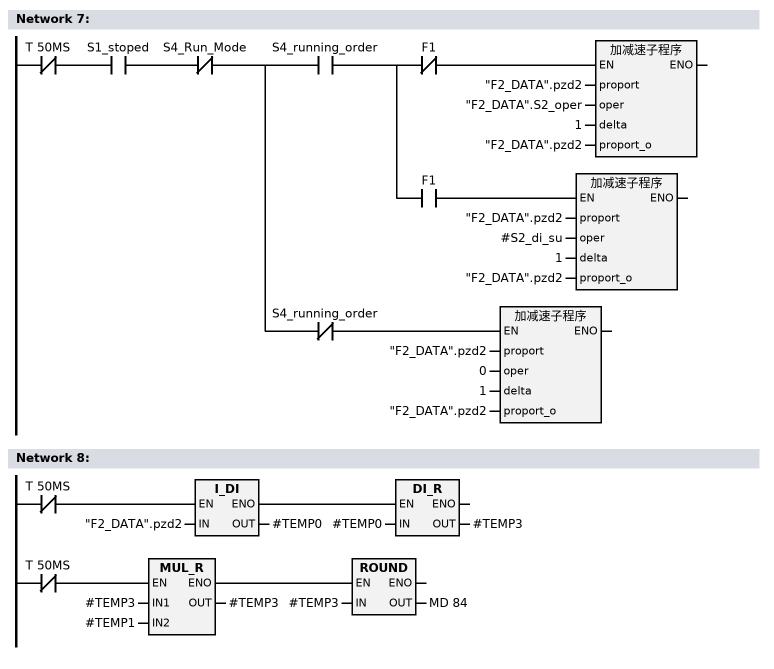
NETWORK
TITLE =
      AN    "T 50MS";
      A     "S1_stoped";
      AN    "S4_Run_Mode";
      =     L 20.0;
      A     L 20.0;
      A     "S4_running_order";
      =     L 20.1;
      A     L 20.1;
      AN    "F1";
      JNB   _00e;
      CALL  "加减速子程序" (
           proport                  := "F2_DATA".pzd2,
           oper                     := "F2_DATA".S2_oper,
           delta                    := 1,
           proport_o                := "F2_DATA".pzd2);
_00e: NOP   0;
      A     L 20.1;
      A     "F1";
      JNB   _00f;
      CALL  "加减速子程序" (
           proport                  := "F2_DATA".pzd2,
           oper                     := #S2_di_su,
           delta                    := 1,
           proport_o                := "F2_DATA".pzd2);
_00f: NOP   0;
      A     L 20.0;
      AN    "S4_running_order";
      JNB   _010;
      CALL  "加减速子程序" (
           proport                  := "F2_DATA".pzd2,
           oper                     := 0,
           delta                    := 1,
           proport_o                := "F2_DATA".pzd2);
_010: NOP   0;
NETWORK
TITLE =
      AN    "T 50MS";
      =     L 20.0;
      A(;
      A     L 20.0;
      JNB   _011;
      L     "F2_DATA".pzd2;
      ITD;
      T     #TEMP0;
      SET;
      SAVE;
      CLR;
_011: A     BR;
      );
      JNB   _012;
      L     #TEMP0;
      DTR;
      T     #TEMP3;
_012: NOP   0;
      A(;
      A     L 20.0;
      JNB   _013;
      L     #TEMP3;
      L     #TEMP1;
      *R;
      T     #TEMP3;
      AN    OV;
      SAVE;
      CLR;
_013: A     BR;
      );
      JNB   _014;
      L     #TEMP3;
      RND;
      T     MD 84;
_014: NOP   0;
END_FUNCTION

FUNCTION FC 114 : VOID
VERSION : 0.1
BEGIN
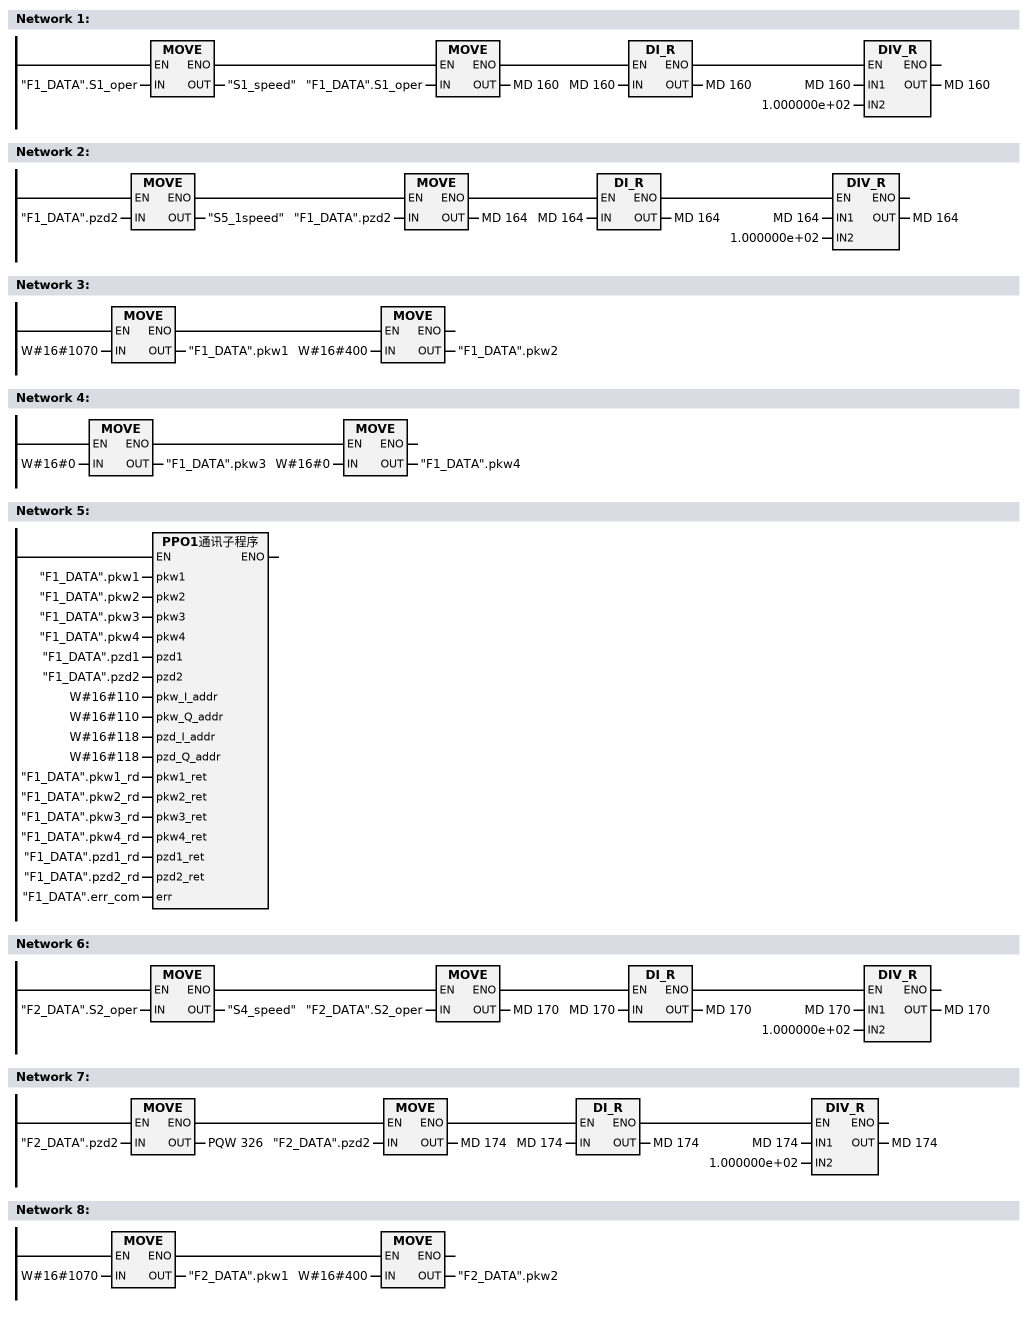
NETWORK
TITLE =
      A(;
      A(;
      A(;
      L     "F1_DATA".S1_oper;
      T     "S1_speed";
      SET;
      SAVE;
      CLR;
      A     BR;
      );
      JNB   _001;
      L     "F1_DATA".S1_oper;
      T     MD 160;
      SET;
      SAVE;
      CLR;
_001: A     BR;
      );
      JNB   _002;
      L     MD 160;
      DTR;
      T     MD 160;
      SET;
      SAVE;
      CLR;
_002: A     BR;
      );
      JNB   _003;
      L     MD 160;
      L     1.000000e+02;
      /R;
      T     MD 160;
_003: NOP   0;
NETWORK
TITLE =
      A(;
      A(;
      A(;
      L     "F1_DATA".pzd2;
      T     "S5_1speed";
      SET;
      SAVE;
      CLR;
      A     BR;
      );
      JNB   _004;
      L     "F1_DATA".pzd2;
      T     MD 164;
      SET;
      SAVE;
      CLR;
_004: A     BR;
      );
      JNB   _005;
      L     MD 164;
      DTR;
      T     MD 164;
      SET;
      SAVE;
      CLR;
_005: A     BR;
      );
      JNB   _006;
      L     MD 164;
      L     1.000000e+02;
      /R;
      T     MD 164;
_006: NOP   0;
NETWORK
TITLE =
      A(;
      L     W#16#1070;
      T     "F1_DATA".pkw1;
      SET;
      SAVE;
      CLR;
      A     BR;
      );
      JNB   _007;
      L     W#16#400;
      T     "F1_DATA".pkw2;
_007: NOP   0;
NETWORK
TITLE =
      A(;
      L     W#16#0;
      T     "F1_DATA".pkw3;
      SET;
      SAVE;
      CLR;
      A     BR;
      );
      JNB   _008;
      L     W#16#0;
      T     "F1_DATA".pkw4;
_008: NOP   0;
NETWORK
TITLE =
      CALL  "PPO1通讯子程序" (
           pkw1                     := "F1_DATA".pkw1,
           pkw2                     := "F1_DATA".pkw2,
           pkw3                     := "F1_DATA".pkw3,
           pkw4                     := "F1_DATA".pkw4,
           pzd1                     := "F1_DATA".pzd1,
           pzd2                     := "F1_DATA".pzd2,
           pkw_I_addr               := W#16#110,
           pkw_Q_addr               := W#16#110,
           pzd_I_addr               := W#16#118,
           pzd_Q_addr               := W#16#118,
           pkw1_ret                 := "F1_DATA".pkw1_rd,
           pkw2_ret                 := "F1_DATA".pkw2_rd,
           pkw3_ret                 := "F1_DATA".pkw3_rd,
           pkw4_ret                 := "F1_DATA".pkw4_rd,
           pzd1_ret                 := "F1_DATA".pzd1_rd,
           pzd2_ret                 := "F1_DATA".pzd2_rd,
           err                      := "F1_DATA".err_com);
      NOP   0;
NETWORK
TITLE =
      A(;
      A(;
      A(;
      L     "F2_DATA".S2_oper;
      T     "S4_speed";
      SET;
      SAVE;
      CLR;
      A     BR;
      );
      JNB   _009;
      L     "F2_DATA".S2_oper;
      T     MD 170;
      SET;
      SAVE;
      CLR;
_009: A     BR;
      );
      JNB   _00a;
      L     MD 170;
      DTR;
      T     MD 170;
      SET;
      SAVE;
      CLR;
_00a: A     BR;
      );
      JNB   _00b;
      L     MD 170;
      L     1.000000e+02;
      /R;
      T     MD 170;
_00b: NOP   0;
NETWORK
TITLE =
      A(;
      A(;
      A(;
      L     "F2_DATA".pzd2;
      T     PQW 326;
      SET;
      SAVE;
      CLR;
      A     BR;
      );
      JNB   _00c;
      L     "F2_DATA".pzd2;
      T     MD 174;
      SET;
      SAVE;
      CLR;
_00c: A     BR;
      );
      JNB   _00d;
      L     MD 174;
      DTR;
      T     MD 174;
      SET;
      SAVE;
      CLR;
_00d: A     BR;
      );
      JNB   _010;
      L     MD 174;
      L     1.000000e+02;
      /R;
      T     MD 174;
_010: NOP   0;
NETWORK
TITLE =
      A(;
      L     W#16#1070;
      T     "F2_DATA".pkw1;
      SET;
      SAVE;
      CLR;
      A     BR;
      );
      JNB   _011;
      L     W#16#400;
      T     "F2_DATA".pkw2;
_011: NOP   0;
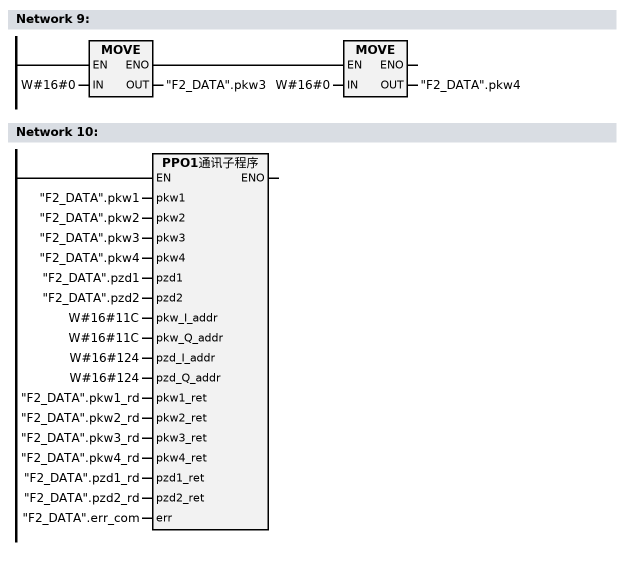
NETWORK
TITLE =
      A(;
      L     W#16#0;
      T     "F2_DATA".pkw3;
      SET;
      SAVE;
      CLR;
      A     BR;
      );
      JNB   _012;
      L     W#16#0;
      T     "F2_DATA".pkw4;
_012: NOP   0;
NETWORK
TITLE =
      CALL  "PPO1通讯子程序" (
           pkw1                     := "F2_DATA".pkw1,
           pkw2                     := "F2_DATA".pkw2,
           pkw3                     := "F2_DATA".pkw3,
           pkw4                     := "F2_DATA".pkw4,
           pzd1                     := "F2_DATA".pzd1,
           pzd2                     := "F2_DATA".pzd2,
           pkw_I_addr               := W#16#11C,
           pkw_Q_addr               := W#16#11C,
           pzd_I_addr               := W#16#124,
           pzd_Q_addr               := W#16#124,
           pkw1_ret                 := "F2_DATA".pkw1_rd,
           pkw2_ret                 := "F2_DATA".pkw2_rd,
           pkw3_ret                 := "F2_DATA".pkw3_rd,
           pkw4_ret                 := "F2_DATA".pkw4_rd,
           pzd1_ret                 := "F2_DATA".pzd1_rd,
           pzd2_ret                 := "F2_DATA".pzd2_rd,
           err                      := "F2_DATA".err_com);
      NOP   0;
END_FUNCTION

DATA_BLOCK "F1_DATA"	// DB 1
VERSION : 0.1
  STRUCT
   pkw1 : WORD  := W#16#1070;
   pkw2 : WORD  := W#16#400;
   pkw3 : WORD ;
   pkw4 : WORD ;
   pzd1 : WORD  := W#16#82;
   pzd2 : INT  := 2000;
   pkw1_rd : WORD ;
   pkw2_rd : WORD ;
   pkw3_rd : WORD ;
   pkw4_rd : WORD ;
   pzd1_rd : WORD ;
   pzd2_rd : WORD ;
   err_com : BOOL ;
   S1_oper : INT ;
  END_STRUCT ;	
BEGIN
   pkw1 := W#16#1070;
   pkw2 := W#16#400;
   pzd1 := W#16#82;
   pzd2 := 2000;
END_DATA_BLOCK

DATA_BLOCK "F2_DATA"	// DB 2
VERSION : 0.1
  STRUCT
   pkw1 : WORD ;
   pkw2 : WORD ;
   pkw3 : WORD ;
   pkw4 : WORD ;
   pzd1 : WORD ;
   pzd2 : INT ;
   pkw1_rd : WORD ;
   pkw2_rd : WORD ;
   pkw3_rd : WORD ;
   pkw4_rd : WORD ;
   pzd1_rd : WORD ;
   pzd2_rd : WORD ;
   err_com : BOOL ;
   S2_oper : INT ;
  END_STRUCT ;	
BEGIN
END_DATA_BLOCK

ORGANIZATION_BLOCK OB 1
TITLE = "Main Program Sweep (Cycle)"
VERSION : 0.1
VAR_TEMP
  OB1_EV_CLASS : BYTE ;	//Bits 0-3 = 1 (Coming event), Bits 4-7 = 1 (Event class 1)
  OB1_SCAN_1 : BYTE ;	//1 (Cold restart scan 1 of OB 1), 3 (Scan 2-n of OB 1)
  OB1_PRIORITY : BYTE ;	//Priority of OB Execution
  OB1_OB_NUMBR : BYTE ;	//1 (Organization block 1, OB1)
  OB1_RESERVED_1 : BYTE ;	//Reserved for system
  OB1_RESERVED_2 : BYTE ;	//Reserved for system
  OB1_PREV_CYCLE : INT ;	//Cycle time of previous OB1 scan (milliseconds)
  OB1_MIN_CYCLE : INT ;	//Minimum cycle time of OB1 (milliseconds)
  OB1_MAX_CYCLE : INT ;	//Maximum cycle time of OB1 (milliseconds)
  OB1_DATE_TIME : DATE_AND_TIME ;	//Date and time OB1 started
END_VAR
BEGIN
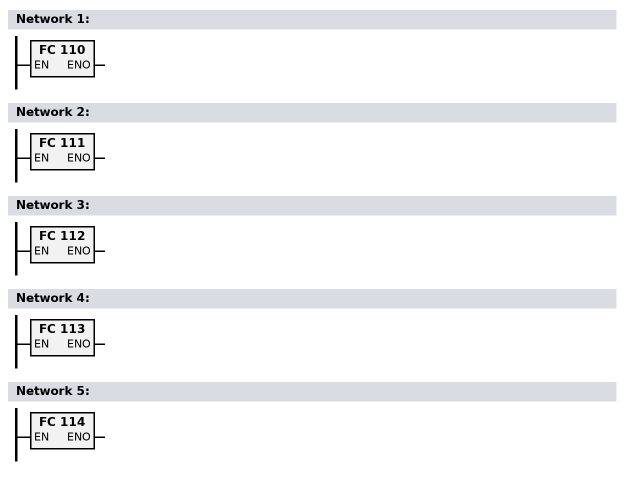
NETWORK
TITLE =
      CALL  FC 110;
      NOP   0;
NETWORK
TITLE =
      CALL  FC 111;
      NOP   0;
NETWORK
TITLE =
      CALL  FC 112;
      NOP   0;
NETWORK
TITLE =
      CALL  FC 113;
      NOP   0;
NETWORK
TITLE =
      CALL  FC 114;
      NOP   0;
END_ORGANIZATION_BLOCK
